// TIA Portal V17 export
// export: Created 2025-03-10T12:17:32.4750853Z, ExportSetting WithDefaults, DisplayName Totally Integrated Automation Portal, DisplayVersion V17 Update 8, DisplayName TIA Portal Openness, DisplayVersion V17 Update 8, DisplayName TIA Portal Version Control Interface, DisplayVersion V17, DisplayName SINAMICS Startdrive Advanced, DisplayVersion V17 SP2, DisplayName SINAMICS Startdrive G110M, G120, G120C, G120D, G120P, G115D, DisplayVersion V17 SP2, DisplayName SINAMICS Startdrive G130, G150, S120, S150, SINAMICS MV, S210, DisplayVersion V17 SP2, DisplayName STEP 7 Professional, DisplayVersion V17 Update 8, DisplayName SINUMERIK ONE STEP 7 Toolbox, DisplayVersion V17 Update 12, DisplayName SINUMERIK 840D sl STEP 7 Toolbox, DisplayVersion V17 Update 12, DisplayName STEP 7 Safety, DisplayVersion V17 Update 6, DisplayName WinCC Advanced, DisplayVersion V17 Update 8
VAR_GLOBAL   // PLC tag table "TAGS_SAFETY_AXES"
   X23_SAFETY_IN AT %I6732.0 : "AXIS_SAFETY_IN";   // CLADDING NCU AXIS 3
   E20_SAFETY_OUT AT %Q6892.0 : "AXIS_SAFETY_OUT";   // CLADDING NX X104 AXIS 13
   C14_SAFETY_IN AT %I6844.0 : "AXIS_SAFETY_IN";   // CLADDING NX X105 AXIS 10
   C14_SAFETY_OUT AT %Q6844.0 : "AXIS_SAFETY_OUT";   // CLADDING NX X105 AXIS 10
   C23_SAFETY_OUT AT %Q6924.0 : "AXIS_SAFETY_OUT";   // CLADDING NX X104 AXIS 15
   UNIT_3_AXES AT %M6796.3 : Bool;
   C22_SAFETY_OUT AT %Q6956.0 : "AXIS_SAFETY_OUT";   // CLADDING NX X104 AXIS 17
   C24_SAFETY_IN AT %I6940.0 : "AXIS_SAFETY_IN";   // CLADDING NX X103 AXIS 16
   C23_SAFETY_IN AT %I6924.0 : "AXIS_SAFETY_IN";   // CLADDING NX X104 AXIS 15
   C12_SAFETY_OUT AT %Q6860.0 : "AXIS_SAFETY_OUT";   // CLADDING NX X105 AXIS 11
   Z11_SAFETY_OUT AT %Q6988.0 : "AXIS_SAFETY_OUT";   // CLADDING NX X102 AXIS 19
   C12_SAFETY_IN AT %I6860.0 : "AXIS_SAFETY_IN";   // CLADDING NX X105 AXIS 11
   Z13_SAFETY_IN AT %I6716.0 : "AXIS_SAFETY_IN";   // CLADDING NCU AXIS 2
   Z13_SAFETY_OUT AT %Q6716.0 : "AXIS_SAFETY_OUT";   // CLADDING NCU AXIS 2
   C13_SAFETY_OUT AT %Q6828.0 : "AXIS_SAFETY_OUT";   // CLADDING NX X105 AXIS 9
   C11_SAFETY_OUT AT %Q6812.0 : "AXIS_SAFETY_OUT";   // CLADDING NX X105 AXIS 8
   C21_SAFETY_OUT AT %Q6908.0 : "AXIS_SAFETY_OUT";   // CLADDING NX X104 AXIS 14
   X13_SAFETY_IN AT %I6700.0 : "AXIS_SAFETY_IN";   // CLADDING NCU AXIS 1
   Z21_SAFETY_IN AT %I7004.0 : "AXIS_SAFETY_IN";   // CLADDING NX X102 AXIS 20
   E10_SAFETY_IN AT %I6796.0 : "AXIS_SAFETY_IN";   // CLADDING NX X105 AXIS 7
   Z21_SAFETY_OUT AT %Q7004.0 : "AXIS_SAFETY_OUT";   // CLADDING NX X102 AXIS 20
   Z23_SAFETY_OUT AT %Q6748.0 : "AXIS_SAFETY_OUT";   // CLADDING NCU AXIS 4
   C24_SAFETY_OUT AT %Q6940.0 : "AXIS_SAFETY_OUT";   // CLADDING NX X103 AXIS 16
   Z11_SAFETY_IN AT %I6988.0 : "AXIS_SAFETY_IN";   // CLADDING NX X102 AXIS 19
   X23_SAFETY_OUT AT %Q6732.0 : "AXIS_SAFETY_OUT";   // CLADDING NCU AXIS 3
   Z23_SAFETY_IN AT %I6748.0 : "AXIS_SAFETY_IN";   // CLADDING NCU AXIS 4
   C11_SAFETY_IN AT %I6812.0 : "AXIS_SAFETY_IN";   // CLADDING NX X105 AXIS 8
   C21_SAFETY_IN AT %I6908.0 : "AXIS_SAFETY_IN";   // CLADDING NX X104 AXIS 14
   C31_SAFETY_OUT AT %Q7020.0 : "AXIS_SAFETY_OUT";   // CLADDING NX X103 AXIS 23
   E10_SAFETY_OUT AT %Q6796.0 : "AXIS_SAFETY_OUT";   // CLADDING NX X105 AXIS 7
   UNIT_2_AXES AT %M6796.2 : Bool;
   C13_SAFETY_IN AT %I6828.0 : "AXIS_SAFETY_IN";   // CLADDING NX X105 AXIS 9
   C31_SAFETY_IN AT %I7020.0 : "AXIS_SAFETY_IN";   // CLADDING NX X103 AXIS 23
   E20_SAFETY_IN AT %I6892.0 : "AXIS_SAFETY_IN";   // CLADDING NX X104 AXIS 13
   UNIT_1_AXES AT %M6796.1 : Bool;
   C22_SAFETY_IN AT %I6956.0 : "AXIS_SAFETY_IN";   // CLADDING NX X104 AXIS 17
   X13_SAFETY_OUT AT %Q6700.0 : "AXIS_SAFETY_OUT";   // CLADDING NCU AXIS 1
END_VAR
